// LS Electric XG5000 project: 크랙 PLC
// PLC NewPLC
// module base 0 slot 0: 입출력 모듈:XBM-DN32H (DC 24V입력/TR 출력, 32점)

PROGRAM NewProgram (task: 스캔 프로그램)

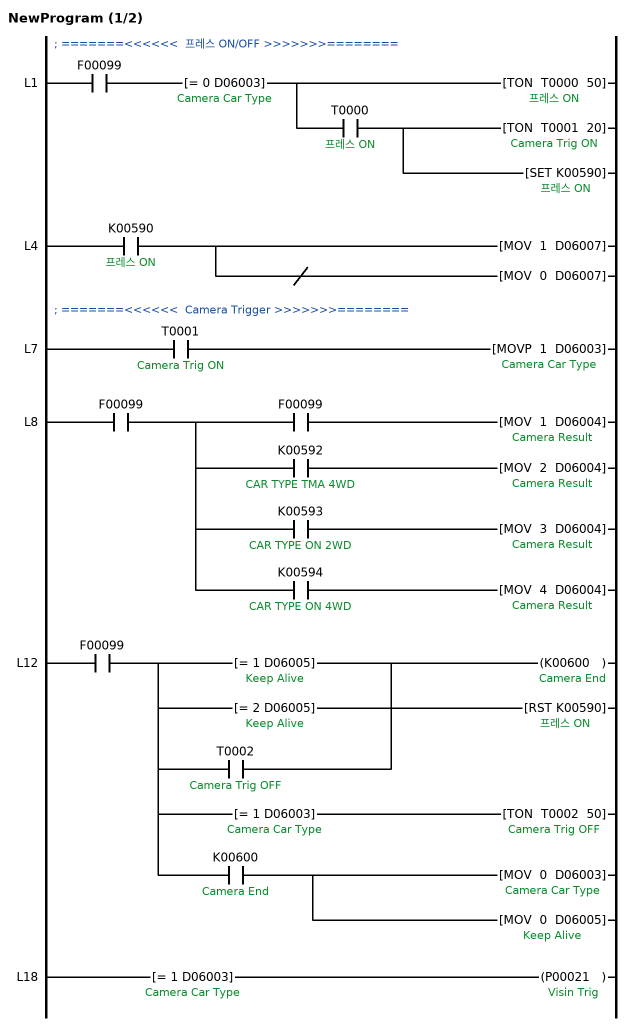
// =======<<<<<<  프레스 ON/OFF >>>>>>>========
; L1
LOAD      F00099
AND=      0 D06003	// Camera Car Type
TON       T0000 50	// 프레스 ON
AND       T0000	// 프레스 ON
TON       T0001 20	// Camera Trig ON
SET       K00590	// 프레스 ON
; L4
LOAD      K00590	// 프레스 ON
MOV       1 D06007
NOT
MOV       0 D06007
// =======<<<<<<  Camera Trigger >>>>>>>========
; L7
LOAD      T0001	// Camera Trig ON
MOVP      1 D06003	// Camera Car Type
; L8
LOAD      F00099
MPUSH
AND       F00099
MOV       1 D06004	// Camera Result
MLOAD
AND       K00592	// CAR TYPE TMA 4WD
MOV       2 D06004	// Camera Result
MLOAD
AND       K00593	// CAR TYPE ON 2WD
MOV       3 D06004	// Camera Result
MPOP
AND       K00594	// CAR TYPE ON 4WD
MOV       4 D06004	// Camera Result
; L12
LOAD      F00099
MPUSH
LOAD=     1 D06005	// Keep Alive
OR=       2 D06005	// Keep Alive
OR        T0002	// Camera Trig OFF
AND LOAD
OUT       K00600	// Camera End
RST       K00590	// 프레스 ON
MLOAD
AND=      1 D06003	// Camera Car Type
TON       T0002 50	// Camera Trig OFF
MPOP
AND       K00600	// Camera End
MOV       0 D06003	// Camera Car Type
MOV       0 D06005	// Keep Alive
; L18
LOAD=     1 D06003	// Camera Car Type
OUT       P00021	// Visin Trig

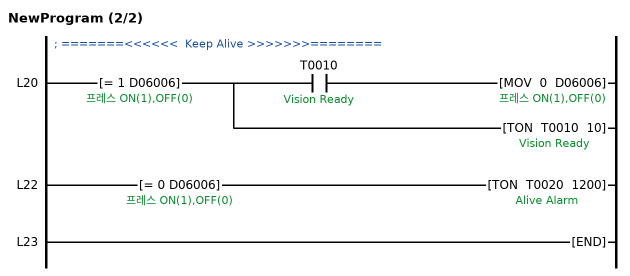
// =======<<<<<<  Keep Alive >>>>>>>========
; L20
LOAD=     1 D06006	// 프레스 ON(1),OFF(0)
MPUSH
AND       T0010	// Vision Ready
MOV       0 D06006	// 프레스 ON(1),OFF(0)
MPOP
TON       T0010 10	// Vision Ready
; L22
LOAD=     0 D06006	// 프레스 ON(1),OFF(0)
TON       T0020 1200	// Alive Alarm
; L23
END

VARIABLES AND COMMENTS (devices not used above)
K00591	BIT	CAR TYPE TMA 2WD
P00020	BIT	OCR Trig
D06002	WORD	Camera Trgger
T0015	BIT/WORD	Camera Reset